(* Visualisation VIS_ANZ
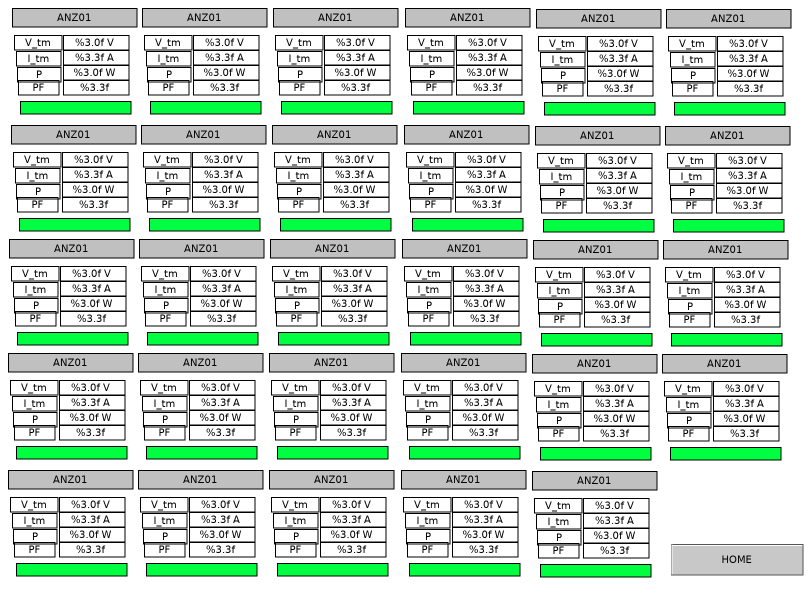
rectangle at (51,38)-(117,53): text "%3.0f V"; shows .ANZ01.Voltage_L1_L2
rectangle at (2,38)-(50,53): text "V_tm"
rectangle at (4,54)-(49,69): text "I_tm"
rectangle at (5,70)-(49,85): text "P"
rectangle at (6,83)-(47,98): text "PF"
rectangle at (51,53)-(117,68): text "%3.3f A"; shows .ANZ01.Current_L1
rectangle at (51,68)-(117,83): text "%3.0f W"; shows .ANZ01.ActivePower
rectangle at (51,83)-(117,98): text "%3.3f"; shows .ANZ01.Power_factor_L1
rectangle at (8,104)-(119,117): alarm colour if .ANZ01.AllarmeNodo
rectangle at (0,11)-(125,30): text "ANZ01"
rectangle at (181,38)-(247,53): text "%3.0f V"; shows .ANZ01.Voltage_L1_L2
rectangle at (132,38)-(180,53): text "V_tm"
rectangle at (134,54)-(179,69): text "I_tm"
rectangle at (135,70)-(179,85): text "P"
rectangle at (136,83)-(177,98): text "PF"
rectangle at (181,53)-(247,68): text "%3.3f A"; shows .ANZ01.Current_L1
rectangle at (181,68)-(247,83): text "%3.0f W"; shows .ANZ01.ActivePower
rectangle at (181,83)-(247,98): text "%3.3f"; shows .ANZ01.Power_factor_L1
rectangle at (138,104)-(249,117): alarm colour if .ANZ01.AllarmeNodo
rectangle at (130,11)-(255,30): text "ANZ01"
rectangle at (312,38)-(378,53): text "%3.0f V"; shows .ANZ01.Voltage_L1_L2
rectangle at (263,38)-(311,53): text "V_tm"
rectangle at (265,54)-(310,69): text "I_tm"
rectangle at (266,70)-(310,85): text "P"
rectangle at (267,83)-(308,98): text "PF"
rectangle at (312,53)-(378,68): text "%3.3f A"; shows .ANZ01.Current_L1
rectangle at (312,68)-(378,83): text "%3.0f W"; shows .ANZ01.ActivePower
rectangle at (312,83)-(378,98): text "%3.3f"; shows .ANZ01.Power_factor_L1
rectangle at (269,104)-(380,117): alarm colour if .ANZ01.AllarmeNodo
rectangle at (261,11)-(386,30): text "ANZ01"
rectangle at (444,38)-(510,53): text "%3.0f V"; shows .ANZ01.Voltage_L1_L2
rectangle at (395,38)-(443,53): text "V_tm"
rectangle at (397,54)-(442,69): text "I_tm"
rectangle at (398,70)-(442,85): text "P"
rectangle at (399,83)-(440,98): text "PF"
rectangle at (444,53)-(510,68): text "%3.3f A"; shows .ANZ01.Current_L1
rectangle at (444,68)-(510,83): text "%3.0f W"; shows .ANZ01.ActivePower
rectangle at (444,83)-(510,98): text "%3.3f"; shows .ANZ01.Power_factor_L1
rectangle at (401,104)-(512,117): alarm colour if .ANZ01.AllarmeNodo
rectangle at (393,11)-(518,30): text "ANZ01"
rectangle at (575,39)-(641,54): text "%3.0f V"; shows .ANZ01.Voltage_L1_L2
rectangle at (526,39)-(574,54): text "V_tm"
rectangle at (528,55)-(573,70): text "I_tm"
rectangle at (529,71)-(573,86): text "P"
rectangle at (530,84)-(571,99): text "PF"
rectangle at (575,54)-(641,69): text "%3.3f A"; shows .ANZ01.Current_L1
rectangle at (575,69)-(641,84): text "%3.0f W"; shows .ANZ01.ActivePower
rectangle at (575,84)-(641,99): text "%3.3f"; shows .ANZ01.Power_factor_L1
rectangle at (532,105)-(643,118): alarm colour if .ANZ01.AllarmeNodo
rectangle at (524,12)-(649,31): text "ANZ01"
rectangle at (705,39)-(771,54): text "%3.0f V"; shows .ANZ01.Voltage_L1_L2
rectangle at (656,39)-(704,54): text "V_tm"
rectangle at (658,55)-(703,70): text "I_tm"
rectangle at (659,71)-(703,86): text "P"
rectangle at (660,84)-(701,99): text "PF"
rectangle at (705,54)-(771,69): text "%3.3f A"; shows .ANZ01.Current_L1
rectangle at (705,69)-(771,84): text "%3.0f W"; shows .ANZ01.ActivePower
rectangle at (705,84)-(771,99): text "%3.3f"; shows .ANZ01.Power_factor_L1
rectangle at (662,105)-(773,118): alarm colour if .ANZ01.AllarmeNodo
rectangle at (654,12)-(779,31): text "ANZ01"
rectangle at (50,155)-(116,170): text "%3.0f V"; shows .ANZ01.Voltage_L1_L2
rectangle at (1,155)-(49,170): text "V_tm"
rectangle at (3,171)-(48,186): text "I_tm"
rectangle at (4,187)-(48,202): text "P"
rectangle at (5,200)-(46,215): text "PF"
rectangle at (50,170)-(116,185): text "%3.3f A"; shows .ANZ01.Current_L1
rectangle at (50,185)-(116,200): text "%3.0f W"; shows .ANZ01.ActivePower
rectangle at (50,200)-(116,215): text "%3.3f"; shows .ANZ01.Power_factor_L1
rectangle at (7,221)-(118,234): alarm colour if .ANZ01.AllarmeNodo
rectangle at (-1,128)-(124,147): text "ANZ01"
rectangle at (180,155)-(246,170): text "%3.0f V"; shows .ANZ01.Voltage_L1_L2
rectangle at (131,155)-(179,170): text "V_tm"
rectangle at (133,171)-(178,186): text "I_tm"
rectangle at (134,187)-(178,202): text "P"
rectangle at (135,200)-(176,215): text "PF"
rectangle at (180,170)-(246,185): text "%3.3f A"; shows .ANZ01.Current_L1
rectangle at (180,185)-(246,200): text "%3.0f W"; shows .ANZ01.ActivePower
rectangle at (180,200)-(246,215): text "%3.3f"; shows .ANZ01.Power_factor_L1
rectangle at (137,221)-(248,234): alarm colour if .ANZ01.AllarmeNodo
rectangle at (129,128)-(254,147): text "ANZ01"
rectangle at (311,155)-(377,170): text "%3.0f V"; shows .ANZ01.Voltage_L1_L2
rectangle at (262,155)-(310,170): text "V_tm"
rectangle at (264,171)-(309,186): text "I_tm"
rectangle at (265,187)-(309,202): text "P"
rectangle at (266,200)-(307,215): text "PF"
rectangle at (311,170)-(377,185): text "%3.3f A"; shows .ANZ01.Current_L1
rectangle at (311,185)-(377,200): text "%3.0f W"; shows .ANZ01.ActivePower
rectangle at (311,200)-(377,215): text "%3.3f"; shows .ANZ01.Power_factor_L1
rectangle at (268,221)-(379,234): alarm colour if .ANZ01.AllarmeNodo
rectangle at (260,128)-(385,147): text "ANZ01"
rectangle at (443,155)-(509,170): text "%3.0f V"; shows .ANZ01.Voltage_L1_L2
rectangle at (394,155)-(442,170): text "V_tm"
rectangle at (396,171)-(441,186): text "I_tm"
rectangle at (397,187)-(441,202): text "P"
rectangle at (398,200)-(439,215): text "PF"
rectangle at (443,170)-(509,185): text "%3.3f A"; shows .ANZ01.Current_L1
rectangle at (443,185)-(509,200): text "%3.0f W"; shows .ANZ01.ActivePower
rectangle at (443,200)-(509,215): text "%3.3f"; shows .ANZ01.Power_factor_L1
rectangle at (400,221)-(511,234): alarm colour if .ANZ01.AllarmeNodo
rectangle at (392,128)-(517,147): text "ANZ01"
rectangle at (574,156)-(640,171): text "%3.0f V"; shows .ANZ01.Voltage_L1_L2
rectangle at (525,156)-(573,171): text "V_tm"
rectangle at (527,172)-(572,187): text "I_tm"
rectangle at (528,188)-(572,203): text "P"
rectangle at (529,201)-(570,216): text "PF"
rectangle at (574,171)-(640,186): text "%3.3f A"; shows .ANZ01.Current_L1
rectangle at (574,186)-(640,201): text "%3.0f W"; shows .ANZ01.ActivePower
rectangle at (574,201)-(640,216): text "%3.3f"; shows .ANZ01.Power_factor_L1
rectangle at (531,222)-(642,235): alarm colour if .ANZ01.AllarmeNodo
rectangle at (523,129)-(648,148): text "ANZ01"
rectangle at (704,156)-(770,171): text "%3.0f V"; shows .ANZ01.Voltage_L1_L2
rectangle at (655,156)-(703,171): text "V_tm"
rectangle at (657,172)-(702,187): text "I_tm"
rectangle at (658,188)-(702,203): text "P"
rectangle at (659,201)-(700,216): text "PF"
rectangle at (704,171)-(770,186): text "%3.3f A"; shows .ANZ01.Current_L1
rectangle at (704,186)-(770,201): text "%3.0f W"; shows .ANZ01.ActivePower
rectangle at (704,201)-(770,216): text "%3.3f"; shows .ANZ01.Power_factor_L1
rectangle at (661,222)-(772,235): alarm colour if .ANZ01.AllarmeNodo
rectangle at (653,129)-(778,148): text "ANZ01"
rectangle at (48,269)-(114,284): text "%3.0f V"; shows .ANZ01.Voltage_L1_L2
rectangle at (-1,269)-(47,284): text "V_tm"
rectangle at (1,285)-(46,300): text "I_tm"
rectangle at (2,301)-(46,316): text "P"
rectangle at (3,314)-(44,329): text "PF"
rectangle at (48,284)-(114,299): text "%3.3f A"; shows .ANZ01.Current_L1
rectangle at (48,299)-(114,314): text "%3.0f W"; shows .ANZ01.ActivePower
rectangle at (48,314)-(114,329): text "%3.3f"; shows .ANZ01.Power_factor_L1
rectangle at (5,335)-(116,348): alarm colour if .ANZ01.AllarmeNodo
rectangle at (-3,242)-(122,261): text "ANZ01"
rectangle at (178,269)-(244,284): text "%3.0f V"; shows .ANZ01.Voltage_L1_L2
rectangle at (129,269)-(177,284): text "V_tm"
rectangle at (131,285)-(176,300): text "I_tm"
rectangle at (132,301)-(176,316): text "P"
rectangle at (133,314)-(174,329): text "PF"
rectangle at (178,284)-(244,299): text "%3.3f A"; shows .ANZ01.Current_L1
rectangle at (178,299)-(244,314): text "%3.0f W"; shows .ANZ01.ActivePower
rectangle at (178,314)-(244,329): text "%3.3f"; shows .ANZ01.Power_factor_L1
rectangle at (135,335)-(246,348): alarm colour if .ANZ01.AllarmeNodo
rectangle at (127,242)-(252,261): text "ANZ01"
rectangle at (309,269)-(375,284): text "%3.0f V"; shows .ANZ01.Voltage_L1_L2
rectangle at (260,269)-(308,284): text "V_tm"
rectangle at (262,285)-(307,300): text "I_tm"
rectangle at (263,301)-(307,316): text "P"
rectangle at (264,314)-(305,329): text "PF"
rectangle at (309,284)-(375,299): text "%3.3f A"; shows .ANZ01.Current_L1
rectangle at (309,299)-(375,314): text "%3.0f W"; shows .ANZ01.ActivePower
rectangle at (309,314)-(375,329): text "%3.3f"; shows .ANZ01.Power_factor_L1
rectangle at (266,335)-(377,348): alarm colour if .ANZ01.AllarmeNodo
rectangle at (258,242)-(383,261): text "ANZ01"
rectangle at (441,269)-(507,284): text "%3.0f V"; shows .ANZ01.Voltage_L1_L2
rectangle at (392,269)-(440,284): text "V_tm"
rectangle at (394,285)-(439,300): text "I_tm"
rectangle at (395,301)-(439,316): text "P"
rectangle at (396,314)-(437,329): text "PF"
rectangle at (441,284)-(507,299): text "%3.3f A"; shows .ANZ01.Current_L1
rectangle at (441,299)-(507,314): text "%3.0f W"; shows .ANZ01.ActivePower
rectangle at (441,314)-(507,329): text "%3.3f"; shows .ANZ01.Power_factor_L1
rectangle at (398,335)-(509,348): alarm colour if .ANZ01.AllarmeNodo
rectangle at (390,242)-(515,261): text "ANZ01"
rectangle at (572,270)-(638,285): text "%3.0f V"; shows .ANZ01.Voltage_L1_L2
rectangle at (523,270)-(571,285): text "V_tm"
rectangle at (525,286)-(570,301): text "I_tm"
rectangle at (526,302)-(570,317): text "P"
rectangle at (527,315)-(568,330): text "PF"
rectangle at (572,285)-(638,300): text "%3.3f A"; shows .ANZ01.Current_L1
rectangle at (572,300)-(638,315): text "%3.0f W"; shows .ANZ01.ActivePower
rectangle at (572,315)-(638,330): text "%3.3f"; shows .ANZ01.Power_factor_L1
rectangle at (529,336)-(640,349): alarm colour if .ANZ01.AllarmeNodo
rectangle at (521,243)-(646,262): text "ANZ01"
rectangle at (702,270)-(768,285): text "%3.0f V"; shows .ANZ01.Voltage_L1_L2
rectangle at (653,270)-(701,285): text "V_tm"
rectangle at (655,286)-(700,301): text "I_tm"
rectangle at (656,302)-(700,317): text "P"
rectangle at (657,315)-(698,330): text "PF"
rectangle at (702,285)-(768,300): text "%3.3f A"; shows .ANZ01.Current_L1
rectangle at (702,300)-(768,315): text "%3.0f W"; shows .ANZ01.ActivePower
rectangle at (702,315)-(768,330): text "%3.3f"; shows .ANZ01.Power_factor_L1
rectangle at (659,336)-(770,349): alarm colour if .ANZ01.AllarmeNodo
rectangle at (651,243)-(776,262): text "ANZ01"
rectangle at (47,383)-(113,398): text "%3.0f V"; shows .ANZ01.Voltage_L1_L2
rectangle at (-2,383)-(46,398): text "V_tm"
rectangle at (0,399)-(45,414): text "I_tm"
rectangle at (1,415)-(45,430): text "P"
rectangle at (2,428)-(43,443): text "PF"
rectangle at (47,398)-(113,413): text "%3.3f A"; shows .ANZ01.Current_L1
rectangle at (47,413)-(113,428): text "%3.0f W"; shows .ANZ01.ActivePower
rectangle at (47,428)-(113,443): text "%3.3f"; shows .ANZ01.Power_factor_L1
rectangle at (4,449)-(115,462): alarm colour if .ANZ01.AllarmeNodo
rectangle at (-4,356)-(121,375): text "ANZ01"
rectangle at (177,383)-(243,398): text "%3.0f V"; shows .ANZ01.Voltage_L1_L2
rectangle at (128,383)-(176,398): text "V_tm"
rectangle at (130,399)-(175,414): text "I_tm"
rectangle at (131,415)-(175,430): text "P"
rectangle at (132,428)-(173,443): text "PF"
rectangle at (177,398)-(243,413): text "%3.3f A"; shows .ANZ01.Current_L1
rectangle at (177,413)-(243,428): text "%3.0f W"; shows .ANZ01.ActivePower
rectangle at (177,428)-(243,443): text "%3.3f"; shows .ANZ01.Power_factor_L1
rectangle at (134,449)-(245,462): alarm colour if .ANZ01.AllarmeNodo
rectangle at (126,356)-(251,375): text "ANZ01"
rectangle at (308,383)-(374,398): text "%3.0f V"; shows .ANZ01.Voltage_L1_L2
rectangle at (259,383)-(307,398): text "V_tm"
rectangle at (261,399)-(306,414): text "I_tm"
rectangle at (262,415)-(306,430): text "P"
rectangle at (263,428)-(304,443): text "PF"
rectangle at (308,398)-(374,413): text "%3.3f A"; shows .ANZ01.Current_L1
rectangle at (308,413)-(374,428): text "%3.0f W"; shows .ANZ01.ActivePower
rectangle at (308,428)-(374,443): text "%3.3f"; shows .ANZ01.Power_factor_L1
rectangle at (265,449)-(376,462): alarm colour if .ANZ01.AllarmeNodo
rectangle at (257,356)-(382,375): text "ANZ01"
rectangle at (440,383)-(506,398): text "%3.0f V"; shows .ANZ01.Voltage_L1_L2
rectangle at (391,383)-(439,398): text "V_tm"
rectangle at (393,399)-(438,414): text "I_tm"
rectangle at (394,415)-(438,430): text "P"
rectangle at (395,428)-(436,443): text "PF"
rectangle at (440,398)-(506,413): text "%3.3f A"; shows .ANZ01.Current_L1
rectangle at (440,413)-(506,428): text "%3.0f W"; shows .ANZ01.ActivePower
rectangle at (440,428)-(506,443): text "%3.3f"; shows .ANZ01.Power_factor_L1
rectangle at (397,449)-(508,462): alarm colour if .ANZ01.AllarmeNodo
rectangle at (389,356)-(514,375): text "ANZ01"
rectangle at (571,384)-(637,399): text "%3.0f V"; shows .ANZ01.Voltage_L1_L2
rectangle at (522,384)-(570,399): text "V_tm"
rectangle at (524,400)-(569,415): text "I_tm"
rectangle at (525,416)-(569,431): text "P"
rectangle at (526,429)-(567,444): text "PF"
rectangle at (571,399)-(637,414): text "%3.3f A"; shows .ANZ01.Current_L1
rectangle at (571,414)-(637,429): text "%3.0f W"; shows .ANZ01.ActivePower
rectangle at (571,429)-(637,444): text "%3.3f"; shows .ANZ01.Power_factor_L1
rectangle at (528,450)-(639,463): alarm colour if .ANZ01.AllarmeNodo
rectangle at (520,357)-(645,376): text "ANZ01"
rectangle at (701,384)-(767,399): text "%3.0f V"; shows .ANZ01.Voltage_L1_L2
rectangle at (652,384)-(700,399): text "V_tm"
rectangle at (654,400)-(699,415): text "I_tm"
rectangle at (655,416)-(699,431): text "P"
rectangle at (656,429)-(697,444): text "PF"
rectangle at (701,399)-(767,414): text "%3.3f A"; shows .ANZ01.Current_L1
rectangle at (701,414)-(767,429): text "%3.0f W"; shows .ANZ01.ActivePower
rectangle at (701,429)-(767,444): text "%3.3f"; shows .ANZ01.Power_factor_L1
rectangle at (658,450)-(769,463): alarm colour if .ANZ01.AllarmeNodo
rectangle at (650,357)-(775,376): text "ANZ01"
rectangle at (47,500)-(113,515): text "%3.0f V"; shows .ANZ01.Voltage_L1_L2
rectangle at (-2,500)-(46,515): text "V_tm"
rectangle at (0,516)-(45,531): text "I_tm"
rectangle at (1,532)-(45,547): text "P"
rectangle at (2,545)-(43,560): text "PF"
rectangle at (47,515)-(113,530): text "%3.3f A"; shows .ANZ01.Current_L1
rectangle at (47,530)-(113,545): text "%3.0f W"; shows .ANZ01.ActivePower
rectangle at (47,545)-(113,560): text "%3.3f"; shows .ANZ01.Power_factor_L1
rectangle at (4,566)-(115,579): alarm colour if .ANZ01.AllarmeNodo
rectangle at (-4,473)-(121,492): text "ANZ01"
rectangle at (177,500)-(243,515): text "%3.0f V"; shows .ANZ01.Voltage_L1_L2
rectangle at (128,500)-(176,515): text "V_tm"
rectangle at (130,516)-(175,531): text "I_tm"
rectangle at (131,532)-(175,547): text "P"
rectangle at (132,545)-(173,560): text "PF"
rectangle at (177,515)-(243,530): text "%3.3f A"; shows .ANZ01.Current_L1
rectangle at (177,530)-(243,545): text "%3.0f W"; shows .ANZ01.ActivePower
rectangle at (177,545)-(243,560): text "%3.3f"; shows .ANZ01.Power_factor_L1
rectangle at (134,566)-(245,579): alarm colour if .ANZ01.AllarmeNodo
rectangle at (126,473)-(251,492): text "ANZ01"
rectangle at (308,500)-(374,515): text "%3.0f V"; shows .ANZ01.Voltage_L1_L2
rectangle at (259,500)-(307,515): text "V_tm"
rectangle at (261,516)-(306,531): text "I_tm"
rectangle at (262,532)-(306,547): text "P"
rectangle at (263,545)-(304,560): text "PF"
rectangle at (308,515)-(374,530): text "%3.3f A"; shows .ANZ01.Current_L1
rectangle at (308,530)-(374,545): text "%3.0f W"; shows .ANZ01.ActivePower
rectangle at (308,545)-(374,560): text "%3.3f"; shows .ANZ01.Power_factor_L1
rectangle at (265,566)-(376,579): alarm colour if .ANZ01.AllarmeNodo
rectangle at (257,473)-(382,492): text "ANZ01"
rectangle at (440,500)-(506,515): text "%3.0f V"; shows .ANZ01.Voltage_L1_L2
rectangle at (391,500)-(439,515): text "V_tm"
rectangle at (393,516)-(438,531): text "I_tm"
rectangle at (394,532)-(438,547): text "P"
rectangle at (395,545)-(436,560): text "PF"
rectangle at (440,515)-(506,530): text "%3.3f A"; shows .ANZ01.Current_L1
rectangle at (440,530)-(506,545): text "%3.0f W"; shows .ANZ01.ActivePower
rectangle at (440,545)-(506,560): text "%3.3f"; shows .ANZ01.Power_factor_L1
rectangle at (397,566)-(508,579): alarm colour if .ANZ01.AllarmeNodo
rectangle at (389,473)-(514,492): text "ANZ01"
rectangle at (571,501)-(637,516): text "%3.0f V"; shows .ANZ01.Voltage_L1_L2
rectangle at (522,501)-(570,516): text "V_tm"
rectangle at (524,517)-(569,532): text "I_tm"
rectangle at (525,533)-(569,548): text "P"
rectangle at (526,546)-(567,561): text "PF"
rectangle at (571,516)-(637,531): text "%3.3f A"; shows .ANZ01.Current_L1
rectangle at (571,531)-(637,546): text "%3.0f W"; shows .ANZ01.ActivePower
rectangle at (571,546)-(637,561): text "%3.3f"; shows .ANZ01.Power_factor_L1
rectangle at (528,567)-(639,580): alarm colour if .ANZ01.AllarmeNodo
rectangle at (520,474)-(645,493): text "ANZ01"
button at (659,547)-(791,578): text "HOME"; opens PLC_VISU
29 more shapes without text or variables
*)
